{attribute 'linkalways'}
{attribute 'no_explicit_call' := 'This FB is a CLASS and must be accessed using methods or properties'}
{attribute 'enable_dynamic_creation'}
FUNCTION_BLOCK _ETcVnComparisonOperator EXTENDS EnumDatatypeBase
VAR
	localData : ETcVnComparisonOperator;
	activeData : REFERENCE TO ETcVnComparisonOperator;
	enumBaseDatatype : _INT(localData);
END_VAR

METHOD PRIVATE AddLocalEnumeration
VAR_INPUT
	Enumeration : T_MAXSTRING;
	Value : ETcVnComparisonOperator;
END_VAR
AddEnumeration(Enumeration, Value);
END_METHOD

PROPERTY PUBLIC Address : PVOID
GET
Address := ADR(activeData);
END_GET
END_PROPERTY

METHOD PUBLIC ClearReference
VAR_INPUT
END_VAR
activeData REF= localData;
SetBaseDatatypeReference();
END_METHOD

METHOD PUBLIC Clone : I_Datatype
VAR
    pClone : POINTER TO _ETcVnComparisonOperator;
END_VAR
pClone := __NEW(_ETcVnComparisonOperator(InitialValue := Value));
IF pClone = 0 THEN
    RETURN;
END_IF
Clone := pClone^;
END_METHOD

METHOD FB_init : BOOL
VAR_INPUT
	bInitRetains : BOOL; // if TRUE, the retain variables are initialized (warm start / cold start)
	bInCopyCode : BOOL;  // if TRUE, the instance afterwards gets moved into the copy code (online change)
	InitialValue : ETcVnComparisonOperator;
END_VAR
localData := InitialValue;
AddBaseDatatype(enumBaseDatatype);
ClearReference();

AddLocalEnumeration('TCVN_CO_LESS', ETcVnComparisonOperator.TCVN_CO_LESS);
AddLocalEnumeration('TCVN_CO_GREATER', ETcVnComparisonOperator.TCVN_CO_GREATER);
END_METHOD

PROPERTY PUBLIC Identifier : T_MAXSTRING
GET
Identifier := 'ETcVnComparisonOperator';
END_GET
END_PROPERTY

METHOD IsEnumeratorValueEqual : BOOL
VAR_INPUT
	Enumerator : I_KeyValueForwardEnumerator;
END_VAR
VAR
	storedValue : ETcVnComparisonOperator;
END_VAR
IF NOT Enumerator.TryGet(storedValue) THEN
	RETURN;
END_IF

IsEnumeratorValueEqual := storedValue = activeData;
END_METHOD

METHOD PUBLIC MakeReferenceTo
VAR_INPUT
	ReferenceTarget : REFERENCE TO ETcVnComparisonOperator;
END_VAR
activeData REF= ReferenceTarget;
SetBaseDatatypeReference();
END_METHOD

METHOD PROTECTED SetBaseDatatypeReference
VAR_INPUT
END_VAR
enumBaseDatatype.MakeReferenceTo(activeData);
END_METHOD

PROPERTY PUBLIC Size : UDINT
GET
Size := SIZEOF(activeData);
END_GET
END_PROPERTY

METHOD TryMakeReferenceTo : BOOL
VAR_INPUT
	Target : I_Datatype;
END_VAR
VAR
	pTargetData : POINTER TO ETcVnComparisonOperator;
END_VAR
IF NOT IsEquivalentTo(Target) THEN
	RETURN;
END_IF

pTargetData := Target.Address;
activeData REF= pTargetData^;
SetBaseDatatypeReference();
TryMakeReferenceTo := TRUE;
END_METHOD

PROPERTY PUBLIC Value : ETcVnComparisonOperator
GET
Value := activeData;
END_GET
SET
activeData := Value;
END_SET
END_PROPERTY

END_FUNCTION_BLOCK

(* stored: Version 1.1.0.1, ProductVersion 3.1.4026.13
   POU _ETcVnComparisonOperator: Id {aaf22bb9-4ed1-4ae4-a413-ad53216d064d}, SpecialFunc None
   Folder Core: Id {56701f13-c821-4061-a63b-38e1cf741c0a}
   Folder Protected: Id {13dd2602-8b22-4465-906e-b4ba16565681}
   Folder Customize: Id {319ffa53-ef1d-412b-9863-e6fde5159bcd}
   Folder Constructor: Id {5540508d-45ad-4b21-b291-8d080493c109}
   Folder Private: Id {83a96139-e2dd-47a7-a3a5-5d0c5881ac5a}
   Folder Protected: Id {9a3bc1fc-081c-4fa7-9f95-0cedce992a20}
   Method AddLocalEnumeration: Id {1daa0a9c-58d8-4f73-8bc3-6586be4caac6}
   Property Address: Id {ecaf3c42-1aec-4bd0-8c5c-29e712d98f8b}
   Get Get: Id {d6c03b68-9634-4315-9072-cbd8ee7ab698}
   Method ClearReference: Id {058cf179-14a1-4bb0-b339-deafd24c59e8}
   Method Clone: Id {2d7c707d-cc59-4735-a3c0-e65646417a72}
   Method FB_init: Id {b9b48c64-6480-43e6-ac98-4a3ba8d93ea1}
   Property Identifier: Id {dfda2f81-b0f0-408c-a551-8cab41bd9c7f}
   Get Get: Id {94b14a66-67f7-4ecd-b572-6d32cd159633}
   Method IsEnumeratorValueEqual: Id {860b2f6b-8f77-4124-ae5e-59ce09f3d36d}
   Method MakeReferenceTo: Id {5ce0d70a-296f-43a3-bf8a-ab2af06673d9}
   Method SetBaseDatatypeReference: Id {cb24432c-d0da-4d41-8ce7-251e784e0327}
   Property Size: Id {0d46c9a8-e1ad-48d5-9e0c-7b7b00380e21}
   Get Get: Id {68622410-dab8-4415-8905-6fd3f8655d21}
   Method TryMakeReferenceTo: Id {fd256861-20d4-47f7-9738-8a62d6fef4b4}
   Property Value: Id {7726235a-0903-4383-9f98-60ab6faf1f3b}
   Get Get: Id {059b3b8f-32fc-46ea-8b6f-2bc6c2034b9e}
   Set Set: Id {e5657b2c-373e-42c9-9cff-4679ce6a4501} *)
